// TIA Portal V20 export
TYPE "LWONIK_typeSafetyZoneManualOperation"
// stored: Access Published
   STRUCT
      autoStartEnable : Bool;
      doorLockEnable : Bool;
      doorUnlockEnable : Bool;
      rc_AutoEnable : Bool;
      rc_RollChangeEnable : Bool;
      rc_DoorLockEnable : Bool;
      rc_DoorUnlockEnable : Bool;
      hmiOperationEnable : Bool;
      phmiOperationEnable : Bool;
   END_STRUCT;
END_TYPE
